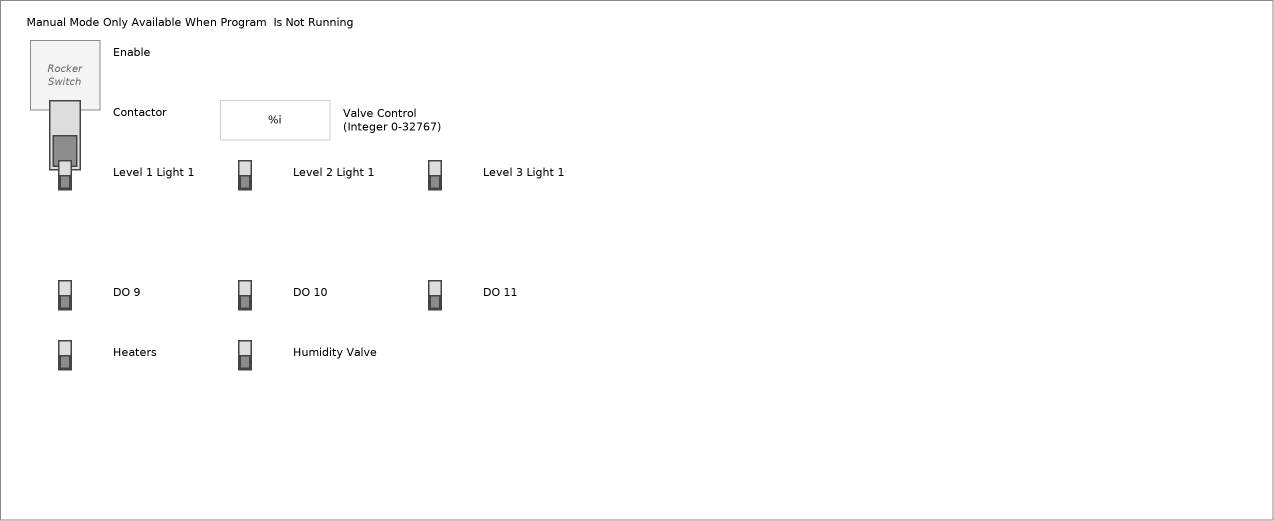
VISUALIZATION ManualMode  // 1274x521
    Label (10,10 360x25), "Manual Mode Only Available When Program Is Not Running"
    RockerSwitch (30,40 70x70), variable: GVL.manualMode, input disabled if: GVL.HMIPowerButton, behaviour: TOGGLE, style: Switch-RockerSwitch-Gray
    DipSwitch (30,100 70x70), variable: IO_VARS.ENABLE, behaviour: TOGGLE, style: Switch-DipSwitch-Gray
    Label (110,40 80x25), "Enable"
    Label (110,100 80x25), "Contactor"
    Label (110,160 110x25), "Level 1 Light 1"
    Textfield (220,100 110x40), "%i", text variable: IO_VARS.GLYCOL_VALVE
        OnMouseClick: write the text variable via VisuDialogs.Numpad, min 0, max 32767
    Label (340,100 100x40), "Valve Control (Integer 0-32767)"
    DipSwitch (30,160 70x30), variable: IO_VARS.FL1, behaviour: TOGGLE, style: Switch-DipSwitch-Gray
    Label (290,160 110x25), "Level 2 Light 1"
    DipSwitch (210,160 70x30), variable: IO_VARS.FL2, behaviour: TOGGLE, style: Switch-DipSwitch-Gray
    Label (480,160 110x25), "Level 3 Light 1"
    DipSwitch (400,160 70x30), variable: IO_VARS.FL3, behaviour: TOGGLE, style: Switch-DipSwitch-Gray
    Label (110,280 110x25), "DO 9"
    DipSwitch (30,280 70x30), variable: IO_VARS.AUX1, behaviour: TOGGLE, style: Switch-DipSwitch-Gray
    Label (290,280 110x25), "DO 10"
    DipSwitch (210,280 70x30), variable: IO_VARS.AUX2, behaviour: TOGGLE, style: Switch-DipSwitch-Gray
    Label (480,280 110x25), "DO 11"
    DipSwitch (400,280 70x30), variable: IO_VARS.AUX3, behaviour: TOGGLE, style: Switch-DipSwitch-Gray
    Label (110,340 110x25), "Heaters"
    DipSwitch (30,340 70x30), variable: IO_VARS.HEATERS, behaviour: TOGGLE, style: Switch-DipSwitch-Gray
    Label (290,340 110x25), "Humidity Valve"
    DipSwitch (210,340 70x30), variable: IO_VARS.HUMVALVE, behaviour: TOGGLE, style: Switch-DipSwitch-Gray
END_VISUALIZATION

(* stored: Version 1.1.0.1, ProductVersion 3.1.4022.18
   Visu ManualMode: Id {4f64843a-1f26-4f8f-be3a-899239e2348d} *)
